KUKA KRL program: C3_HvR.src

&ACCESS RV
&PARAM EDITMASK = *
DEFFCT INT C3_HvR( )

   RETURN 1
ENDFCT
